{attribute 'linkalways'} 
{attribute 'no_explicit_call' := 'This FB is a CLASS and must be accessed using methods or properties'}
{attribute 'enable_dynamic_creation'}
FUNCTION_BLOCK Node_F_VN_CreateHighpassGaussianFilter EXTENDS VisionNode
VAR
    ipFilter : _ITcVnImage;
    nWidth : _UDINT(2);
    nHeight : _UDINT(2);
    bDoublePrecision : _BOOL(FALSE);
    bOriginAtCenter : _BOOL(FALSE);
    fCutoffDistance : _LREAL(1.0);
    hrPrev : _HRESULT(S_OK);
	hresult : _HRESULT(S_OK);
END_VAR

METHOD PUBLIC  Clone : I_Node
VAR
	pNode : POINTER TO Node_F_VN_CreateHighpassGaussianFilter;
END_VAR
pNode := __NEW(Node_F_VN_CreateHighpassGaussianFilter);
Clone := pNode^;
END_METHOD

METHOD FB_init : BOOL
VAR_INPUT
	bInitRetains : BOOL; // if TRUE, the retain variables are initialized (warm start / cold start)
	bInCopyCode : BOOL;  // if TRUE, the instance afterwards gets moved into the copy code (online change)
END_VAR
AddParameter('nWidth', nWidth);
AddParameter('nHeight', nHeight);
AddParameter('bDoublePrecision', bDoublePrecision);
AddParameter('bOriginAtCenter', bOriginAtCenter);
AddParameter('fCutoffDistance', fCutoffDistance);
AddInput('hrPrev', hrPrev);
AddOutput('ipFilter', ipFilter);
AddOutput('hresult',hresult);
END_METHOD

METHOD PROTECTED OnExecute
hresult.Value := F_VN_CreateHighpassGaussianFilter(
    ipFilter := ipFilter.Value,
	nWidth := nWidth.Value,
    nHeight := nHeight.Value,
    bDoublePrecision := bDoublePrecision.Value,
    bOriginAtCenter := bOriginAtCenter.Value,
    fCutoffDistance := fCutoffDistance.Value,
	hrPrev:= hrPrev.Value);
END_METHOD

METHOD PUBLIC PreExecutionCheck
VAR_INPUT
	Check : I_PreExecutionChecks;
END_VAR
Check.IsTrue(nWidth.IsEven, 'nWidth must be an even number');
Check.IsTrue(nHeight.IsEven, 'nHeight must be an even number');
Check.IsTrue((nWidth.Value >= 2), 'nWidth must be greater than or equal to 2');
Check.IsTrue((nHeight.Value >= 2), 'nWidth must be greater than or equal to 2');
Check.IsTrue((fCutoffDistance.Value > 0), 'nCutoffDistance must be greater than 0');
END_METHOD

END_FUNCTION_BLOCK

(* stored: Version 1.1.0.1, ProductVersion 3.1.4024.13
   POU Node_F_VN_CreateHighpassGaussianFilter: Id {d9f9155f-6e4b-06b0-2fd4-3711a0c6aebf}, SpecialFunc None
   Folder Constructor: Id {b546fa20-e4c2-0dfd-3948-1b86f11a915d}
   Method Clone: Id {59ae4bdf-6a56-063a-19f0-e9ab4834e5d4}
   Method FB_init: Id {14a70231-54dc-0460-11f2-3029b86dec4f}
   Method OnExecute: Id {3de562f1-9041-0a9d-08c9-198353bc98c7}
   Method PreExecutionCheck: Id {42c9232a-85f6-0398-0208-7a5dacf4f01f} *)
